// SIMATIC STEP 7 (V5.x) project Practice Project
// CPU: CPU 315-2 DP
// station: Hardware
// station: SIMATIC 300(1)
// station: P_ADR_BUS
// program: S7 Program(1)

SYMBOL_TABLE
"Machine1"	DB 1	DB 1
"Machine2"	DB 2	DB 2
"Counter"	DB 3	DB 3
"Input"	DB 4	DB 4
"Output"	DB 5	DB 5
"Star_Delta"	DB 20	FB 1
"Inpput"	FC 2	FC 2
"Outpput"	FC 3	FC 3
"Logix"	FC 4	FC 4
"SCALE"	FC 105	FC 105	// Scaling Values
"UNSCALE"	FC 106	FC 106	// Unscaling Values
"Start"	I 0.0	BOOL
"Stop"	I 0.1	BOOL
"ON_Switch"	I 4.0	BOOL
"OFF_Switch"	I 4.1	BOOL
"Over_load"	I 4.2	BOOL
"Star_ON"	I 4.3	BOOL
"Star_NC"	I 4.4	BOOL
"Delta_NO"	I 4.5	BOOL
"Delta_NC"	I 4.6	BOOL
"CYCL_EXC"	OB 1	OB 1	// Cycle EXecution
"Motor"	Q 0.0	BOOL
"Main_MC"	Q 4.0	BOOL
"Star_MC"	Q 4.1	BOOL
"Delta_MC"	Q 4.2	BOOL
"Trip_Ind"	Q 4.3	BOOL
"Oven"	UDT 1	UDT 1
"DG"	UDT 2	UDT 2
"VAT_1"	VAT 1	
END_SYMBOL_TABLE

TYPE "Oven"	// UDT 1
VERSION : 0.1
  STRUCT
   Oven_Start : BOOL ;
   Oven_Stop : BOOL ;
   Oven_Run : BOOL ;
   Oven_TEmp : REAL ;
   Oven_Temp_Low : BOOL ;
   Oven_Temp_High : BOOL ;
  END_STRUCT ;	
END_TYPE

TYPE "DG"	// UDT 2
VERSION : 0.1
  STRUCT
   Start : BOOL ;
   Stop : BOOL ;
   Run : BOOL ;
   Temp : REAL ;
   Oil_level_HI : BOOL ;
   Oil_level_Low : BOOL ;
  END_STRUCT ;	
END_TYPE

FUNCTION_BLOCK FB 1
VERSION : 0.1
VAR_INPUT
  Stop : BOOL ;
  Start : BOOL ;
  TD : TIMER ;
  TV : S5TIME ;
  Emergence : BOOL ;
  Overload : BOOL ;
END_VAR
VAR_OUTPUT
  Star : BOOL ;
  Delta : BOOL ;
  Main : BOOL ;
END_VAR
BEGIN
NETWORK
TITLE =
      AN    #Emergence;
      AN    #Overload;
      AN    #Stop;
      A(;
      O     #Start;
      O     #Main;
      );
      =     L 0.0;
      A     L 0.0;
      L     #TV;
      T     LD 1;
      TAK;
      T     LD 5;
      L     #TD;
      T     LW 9;
      L     LD 5;
      L     LD 1;
      SD    T [LW 9];
      NOP   0;
      NOP   0;
      NOP   0;
      NOP   0;
      A     L 0.0;
      T     LD 1;
      TAK;
      T     LD 5;
      L     #TD;
      T     LW 9;
      L     LD 5;
      L     LD 1;
      AN    T [LW 9];
      =     #Star;
      A     L 0.0;
      T     LD 1;
      TAK;
      T     LD 5;
      L     #TD;
      T     LW 9;
      L     LD 5;
      L     LD 1;
      A     T [LW 9];
      =     #Delta;
      A     L 0.0;
      BLD   102;
      =     #Main;
END_FUNCTION_BLOCK

FUNCTION FC 1 : VOID
VERSION : 0.1
BEGIN
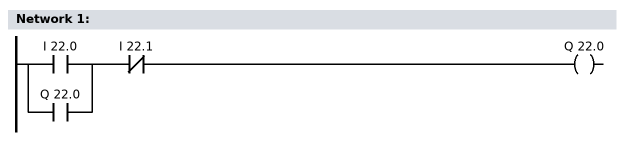
NETWORK
TITLE =
      A(;
      O     I 22.0;
      O     Q 22.0;
      );
      AN    I 22.1;
      =     Q 22.0;
END_FUNCTION

FUNCTION "Inpput" : VOID	// FC 2
VERSION : 0.1
BEGIN
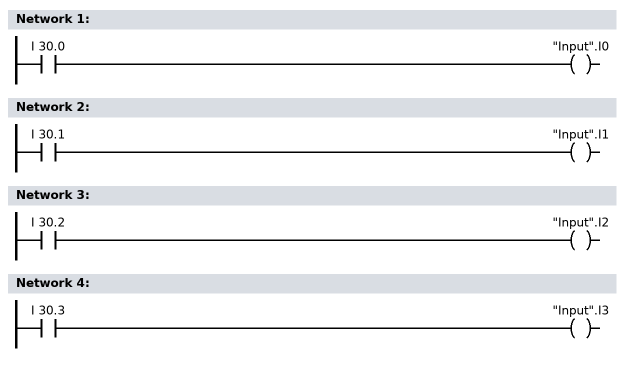
NETWORK
TITLE =
      A     I 30.0;
      =     "Input".I0;
NETWORK
TITLE =
      A     I 30.1;
      =     "Input".I1;
NETWORK
TITLE =
      A     I 30.2;
      =     "Input".I2;
NETWORK
TITLE =
      A     I 30.3;
      =     "Input".I3;
END_FUNCTION

FUNCTION "Outpput" : VOID	// FC 3
VERSION : 0.1
BEGIN
// (block stored without names or comments; labels and parameter names are numbered)
END_FUNCTION

FUNCTION "Logix" : VOID	// FC 4
VERSION : 0.1
BEGIN
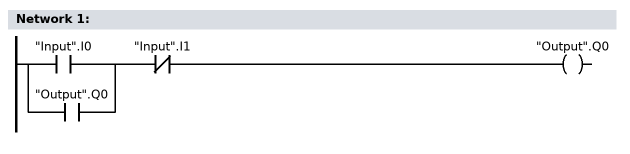
NETWORK
TITLE =
      A(;
      O     "Input".I0;
      O     "Output".Q0;
      );
      AN    "Input".I1;
      =     "Output".Q0;
END_FUNCTION

// FC 105: know-how protected block, not included

// FC 106: know-how protected block, not included

DATA_BLOCK "Machine1"	// DB 1
VERSION : 0.1
  STRUCT
   Start : ARRAY  [1 .. 16 ] OF //Temporary placeholder variable
   BOOL  := FALSE;
   Temp : ARRAY  [1 .. 10 ] OF
   REAL ;
   ADD : ARRAY  [1 .. 100 ] OF DINT ;
   Machine2 : STRUCT
    Start_HMI : BOOL ;
    Stop_HMI : BOOL ;
    Temp1 : REAL ;
    Temp2 : REAL ;
    Generator1 : UDT 2;
    Generator : UDT 2;
    Oven1 : UDT 1;
    Oven2 : UDT 1;
   END_STRUCT ;
  END_STRUCT ;	
BEGIN
END_DATA_BLOCK

DATA_BLOCK "Machine2"	// DB 2
VERSION : 0.1
  STRUCT
   Oven4 : UDT 1;	//Temporary placeholder variable
   Oven5 : UDT 1;
  END_STRUCT ;	
BEGIN
END_DATA_BLOCK

DATA_BLOCK "Counter"	// DB 3
VERSION : 0.1
  STRUCT
   Count : WORD ;	//Temporary placeholder variable
   Count2 : WORD ;
   Count3 : WORD ;
   Count4 : WORD ;
   Sub : ARRAY  [1 .. 10 ] OF INT ;
  END_STRUCT ;	
BEGIN
END_DATA_BLOCK

DATA_BLOCK "Input"	// DB 4
VERSION : 0.1
  STRUCT
   I0 : BOOL ;
   I1 : BOOL ;
   I2 : BOOL ;
   I3 : BOOL ;
   I4 : BOOL ;
   PIW0 : WORD ;
   PIW2 : WORD ;
  END_STRUCT ;	
BEGIN
END_DATA_BLOCK

DATA_BLOCK "Output"	// DB 5
VERSION : 0.1
  STRUCT
   Q0 : BOOL ;
   Q1 : BOOL ;
   Q2 : BOOL ;
   Q3 : BOOL ;
   PQW0 : WORD ;
   PQW2 : WORD ;
  END_STRUCT ;	
BEGIN
END_DATA_BLOCK

DATA_BLOCK "Star_Delta"	// DB 20
VERSION : 0.0
FB 1
BEGIN
END_DATA_BLOCK

DATA_BLOCK DB 21
VERSION : 0.0
FB 1
BEGIN
END_DATA_BLOCK

ORGANIZATION_BLOCK "CYCL_EXC"	// OB 1
TITLE = "Main Program Sweep (Cycle)"
//---------Basic Funcion of various Timer, Converter, Counter etc. 
//Start here------------
VERSION : 0.1
VAR_TEMP
  OB1_EV_CLASS : BYTE ;	//Bits 0-3 = 1 (Coming event), Bits 4-7 = 1 (Event class 1)
  OB1_SCAN_1 : BYTE ;	//1 (Cold restart scan 1 of OB 1), 3 (Scan 2-n of OB 1)
  OB1_PRIORITY : BYTE ;	//Priority of OB Execution
  OB1_OB_NUMBR : BYTE ;	//1 (Organization block 1, OB1)
  OB1_RESERVED_1 : BYTE ;	//Reserved for system
  OB1_RESERVED_2 : BYTE ;	//Reserved for system
  OB1_PREV_CYCLE : INT ;	//Cycle time of previous OB1 scan (milliseconds)
  OB1_MIN_CYCLE : INT ;	//Minimum cycle time of OB1 (milliseconds)
  OB1_MAX_CYCLE : INT ;	//Maximum cycle time of OB1 (milliseconds)
  OB1_DATE_TIME : DATE_AND_TIME ;	//Date and time OB1 started
END_VAR
BEGIN
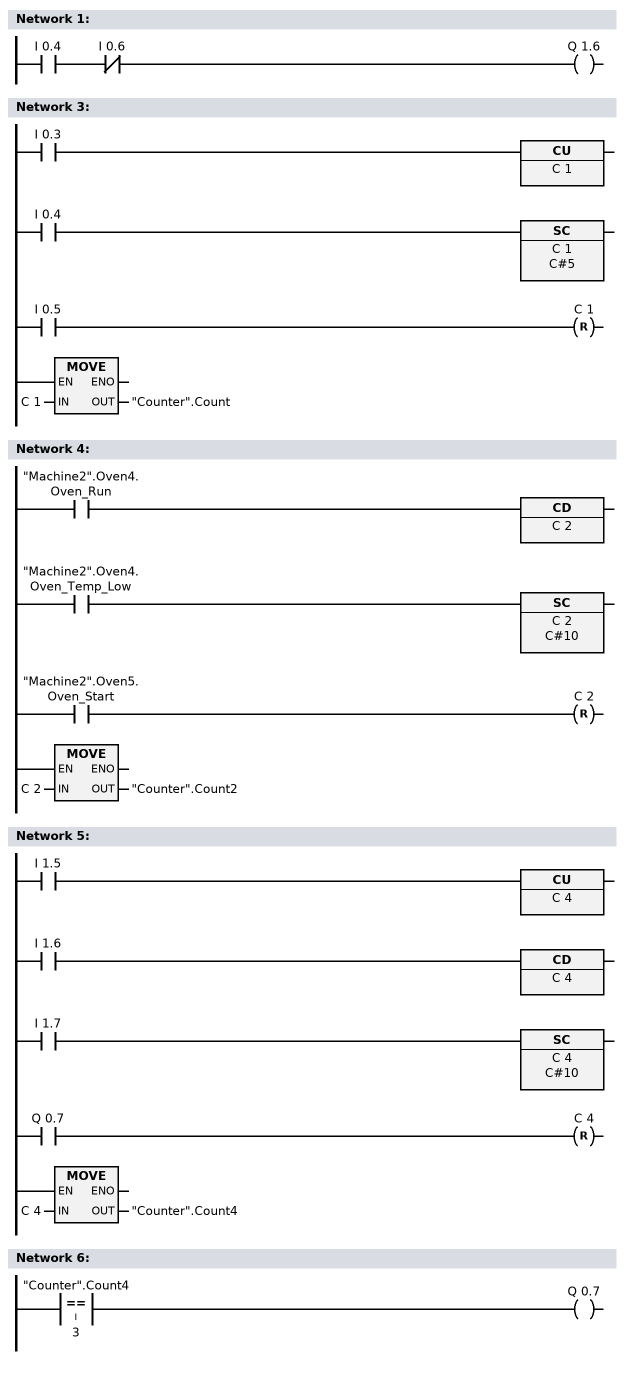
NETWORK
TITLE =
      A     I 0.4;
      AN    I 0.6;
      =     Q 1.6;
NETWORK
TITLE =
NETWORK
TITLE =
      A     I 0.3;
      CU    C 1;
      BLD   101;
      A     I 0.4;
      L     C#5;
      S     C 1;
      A     I 0.5;
      R     C 1;
      L     C 1;
      T     "Counter".Count;
      NOP   0;
      NOP   0;
NETWORK
TITLE =
      A     "Machine2".Oven4.Oven_Run;
      CD    C 2;
      BLD   101;
      A     "Machine2".Oven4.Oven_Temp_Low;
      L     C#10;
      S     C 2;
      A     "Machine2".Oven5.Oven_Start;
      R     C 2;
      L     C 2;
      T     "Counter".Count2;
      NOP   0;
      NOP   0;
NETWORK
TITLE =
      A     I 1.5;
      CU    C 4;
      A     I 1.6;
      CD    C 4;
      A     I 1.7;
      L     C#10;
      S     C 4;
      A     Q 0.7;
      R     C 4;
      L     C 4;
      T     "Counter".Count4;
      NOP   0;
      NOP   0;
NETWORK
TITLE =
      L     "Counter".Count4;
      L     3;
      ==I;
      =     Q 0.7;
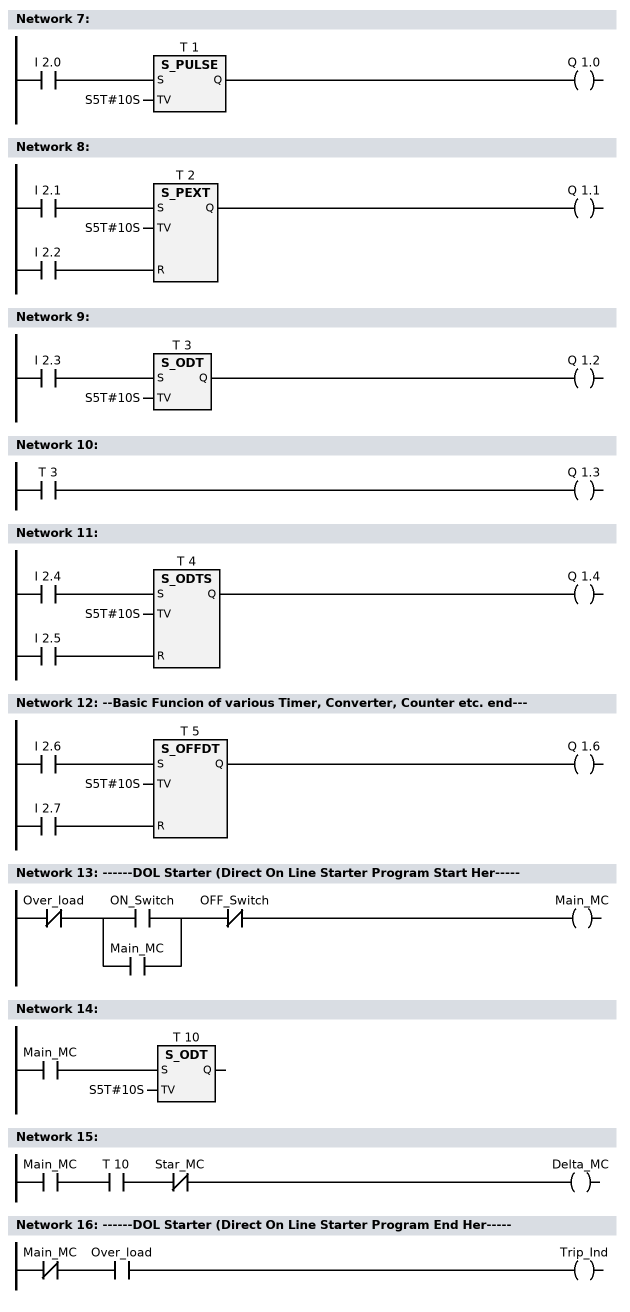
NETWORK
TITLE =
      A     I 2.0;
      L     S5T#10S;
      SP    T 1;
      NOP   0;
      NOP   0;
      NOP   0;
      A     T 1;
      =     Q 1.0;
NETWORK
TITLE =
      A     I 2.1;
      L     S5T#10S;
      SE    T 2;
      A     I 2.2;
      R     T 2;
      NOP   0;
      NOP   0;
      A     T 2;
      =     Q 1.1;
NETWORK
TITLE =
      A     I 2.3;
      L     S5T#10S;
      SD    T 3;
      NOP   0;
      NOP   0;
      NOP   0;
      A     T 3;
      =     Q 1.2;
NETWORK
TITLE =
      A     T 3;
      =     Q 1.3;
NETWORK
TITLE =
      A     I 2.4;
      L     S5T#10S;
      SS    T 4;
      A     I 2.5;
      R     T 4;
      NOP   0;
      NOP   0;
      A     T 4;
      =     Q 1.4;
NETWORK
TITLE = --Basic Funcion of various Timer, Converter, Counter etc. end---
      A     I 2.6;
      L     S5T#10S;
      SF    T 5;
      A     I 2.7;
      R     T 5;
      NOP   0;
      NOP   0;
      A     T 5;
      =     Q 1.6;
NETWORK
TITLE = ------DOL Starter (Direct On Line Starter Program Start Her-----
      AN    "Over_load";
      A(;
      O     "ON_Switch";
      O     "Main_MC";
      );
      AN    "OFF_Switch";
      =     "Main_MC";
NETWORK
TITLE =
      A     "Main_MC";
      L     S5T#10S;
      SD    T 10;
      NOP   0;
      NOP   0;
      NOP   0;
      NOP   0;
NETWORK
TITLE =
      A     "Main_MC";
      A     T 10;
      AN    "Star_MC";
      =     "Delta_MC";
NETWORK
TITLE = ------DOL Starter (Direct On Line Starter Program End Her-----
      AN    "Main_MC";
      A     "Over_load";
      =     "Trip_Ind";
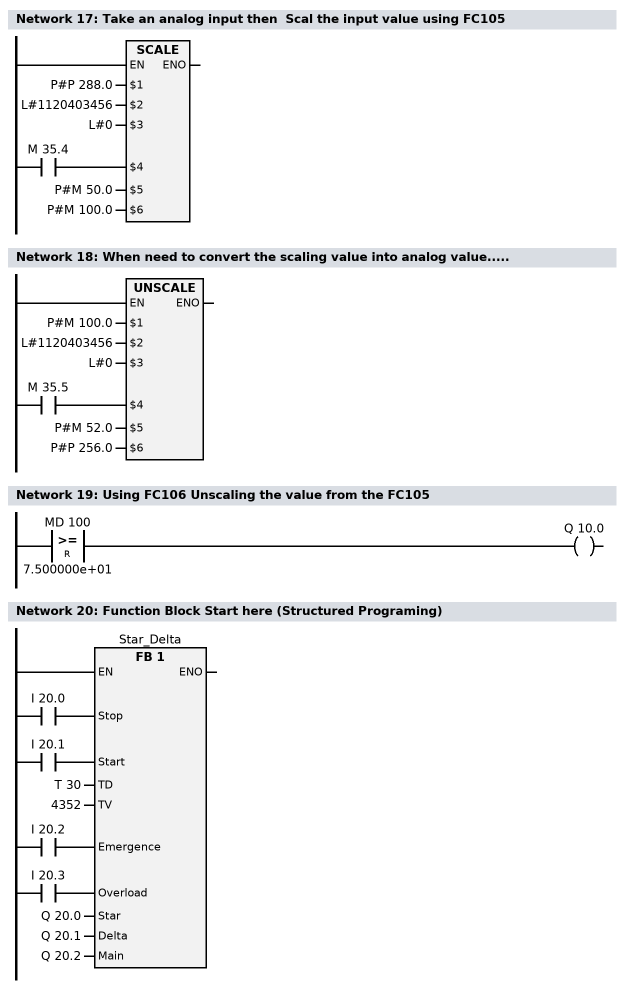
NETWORK
TITLE = Take an analog input then  Scal the input value using FC105
      A     M 35.4;
      =     L 20.0;
      BLD   103;
      CALL  "SCALE" (
           $1                       := P#P 288.0,
           $2                       := L#1120403456,
           $3                       := L#0,
           $4                       := L 20.0,
           $5                       := P#M 50.0,
           $6                       := P#M 100.0);
      NOP   0;
NETWORK
TITLE = When need to convert the scaling value into analog value.....
      A     M 35.5;
      =     L 20.0;
      BLD   103;
      CALL  "UNSCALE" (
           $1                       := P#M 100.0,
           $2                       := L#1120403456,
           $3                       := L#0,
           $4                       := L 20.0,
           $5                       := P#M 52.0,
           $6                       := P#P 256.0);
      NOP   0;
NETWORK
TITLE = Using FC106 Unscaling the value from the FC105 
      L     MD 100;
      L     7.500000e+01;
      >=R;
      =     Q 10.0;
NETWORK
TITLE = Function Block Start here (Structured Programing)
      A     I 20.0;
      =     L 20.0;
      BLD   103;
      A     I 20.1;
      =     L 20.1;
      BLD   103;
      A     I 20.2;
      =     L 20.2;
      BLD   103;
      A     I 20.3;
      =     L 20.3;
      BLD   103;
      CALL  FB 1 , "Star_Delta" (
           Stop                     := L 20.0,
           Start                    := L 20.1,
           TD                       := T 30,
           TV                       := 4352,
           Emergence                := L 20.2,
           Overload                 := L 20.3,
           Star                     := Q 20.0,
           Delta                    := Q 20.1,
           Main                     := Q 20.2);
      NOP   0;
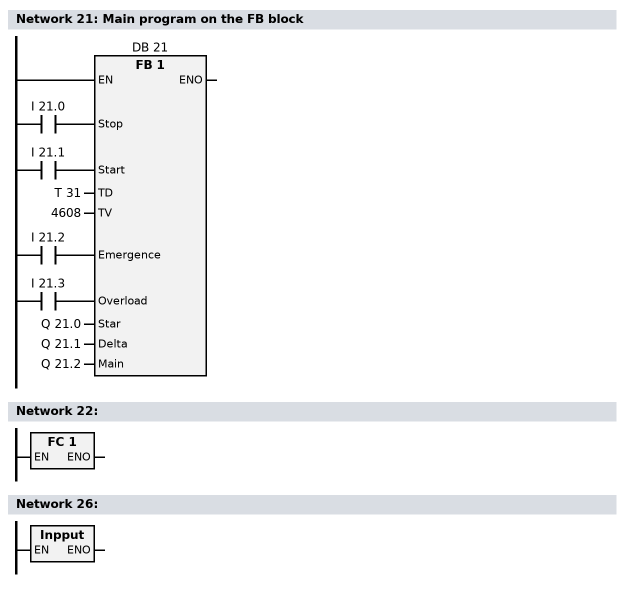
NETWORK
TITLE = Main program on the FB block
      A     I 21.0;
      =     L 20.0;
      BLD   103;
      A     I 21.1;
      =     L 20.1;
      BLD   103;
      A     I 21.2;
      =     L 20.2;
      BLD   103;
      A     I 21.3;
      =     L 20.3;
      BLD   103;
      CALL  FB 1 , DB 21 (
           Stop                     := L 20.0,
           Start                    := L 20.1,
           TD                       := T 31,
           TV                       := 4608,
           Emergence                := L 20.2,
           Overload                 := L 20.3,
           Star                     := Q 21.0,
           Delta                    := Q 21.1,
           Main                     := Q 21.2);
      NOP   0;
NETWORK
TITLE =
      CALL  FC 1;
      NOP   0;
NETWORK
TITLE = Connect input output to the data block(return and call function)
      UC    "Inpput";
NETWORK
TITLE =
      UC    "Logix";
NETWORK
TITLE =
      UC    "Outpput";
NETWORK
TITLE =
      CALL  "Inpput";
      NOP   0;
END_ORGANIZATION_BLOCK
